# EPICS autosave request: profile_bluesky/startup/ref/Db/rebin_settings.req
$(P)rebin$(Q).INPA
$(P)rebin$(Q).INPB
$(P)rebin$(Q).INPC
$(P)rebin$(Q).INPD
$(P)rebin$(Q).INPE
$(P)rebin$(Q).INPF
$(P)rebin$(Q).INPG
